TYPE T_Ctrl_SIf_BCH_Cur :
STRUCT
END_STRUCT
END_TYPE

(* stored: Version 1.1.0.1, ProductVersion 3.1.0.25
   DUT T_Ctrl_SIf_BCH_Cur: Id {9fbe69cb-d086-4801-a109-d65de00c9b31} *)
